// TIA Portal V15.1 export
// export: Created 2024-06-21T08:41:08.5867938Z, ExportSetting WithDefaults, DisplayName Totally Integrated Automation Portal, DisplayVersion V15.1 Update 5, DisplayName TIA Portal Openness, DisplayVersion V15.1 Update 5, DisplayName SINAMICS Startdrive Advanced, DisplayVersion V15.1, DisplayName G130, G150, S120, S150, SINAMICS MV, S210, DisplayVersion V15.1, DisplayName G110M, G120, G120C, G120D, G120P, DisplayVersion V15.1, DisplayName STEP 7 Professional, DisplayVersion V15.1 Update 5, DisplayName STEP 7 Safety, DisplayVersion V15.1, DisplayName WinCC Professional, DisplayVersion V15.1 Update 5, DisplayName SIMATIC Visualization Architect, DisplayVersion V15.1
FUNCTION "LGBJoyStickIAnim" : Void   // FC6612, FBD
TITLE = LIAnimDWord / LGBJoyStickIAnim
{ S7_Optimized_Access := 'TRUE' }
AUTHOR : VCC
FAMILY : Anim
NAME : SIAnim
VERSION : 0.1
// =============================================================================
// Handles the conversion from bits to one Word for simple icon Animation. 
// =============================================================================
// stored: AutoNumber false, IsIECCheckEnabled false, SetENOAutomatically False, UDAEnableTagReadback false
   VAR_INPUT
      I_BtnMiddleAct : Bool;   // Set position / Set Position / Button Middle Active
      I_BtnUpAct : Bool;   // Reset position / Reset Position / Button Up Active
      I_BtnRightAct : Bool;   // Active / Button Right Active
      I_BtnDownAct : Bool;   // ObjectVisible / Button Down Active
      I_BtnLeftAct : Bool;   // Object out of use / Button Left is Active
      I_AnyBtnActive : Bool;   // Any Button Active
      I_OutOfUse : Bool;   // Object out of use
      I_AlarmA : Bool;   // AlarmA
      I_AlarmB : Bool;   // AlarmB
      I_AlarmC : Bool;   // AlarmC
      I_AlarmD : Bool;   // AlarmD
   END_VAR
   VAR_OUTPUT
      H_IAnim : DWord;   // Icon animation Word / Icon Animation
   END_VAR
BEGIN

REGION Network 1: Temporarys output word / **** 1 - Inputs **** Object Out Of Use
   // Object out of use
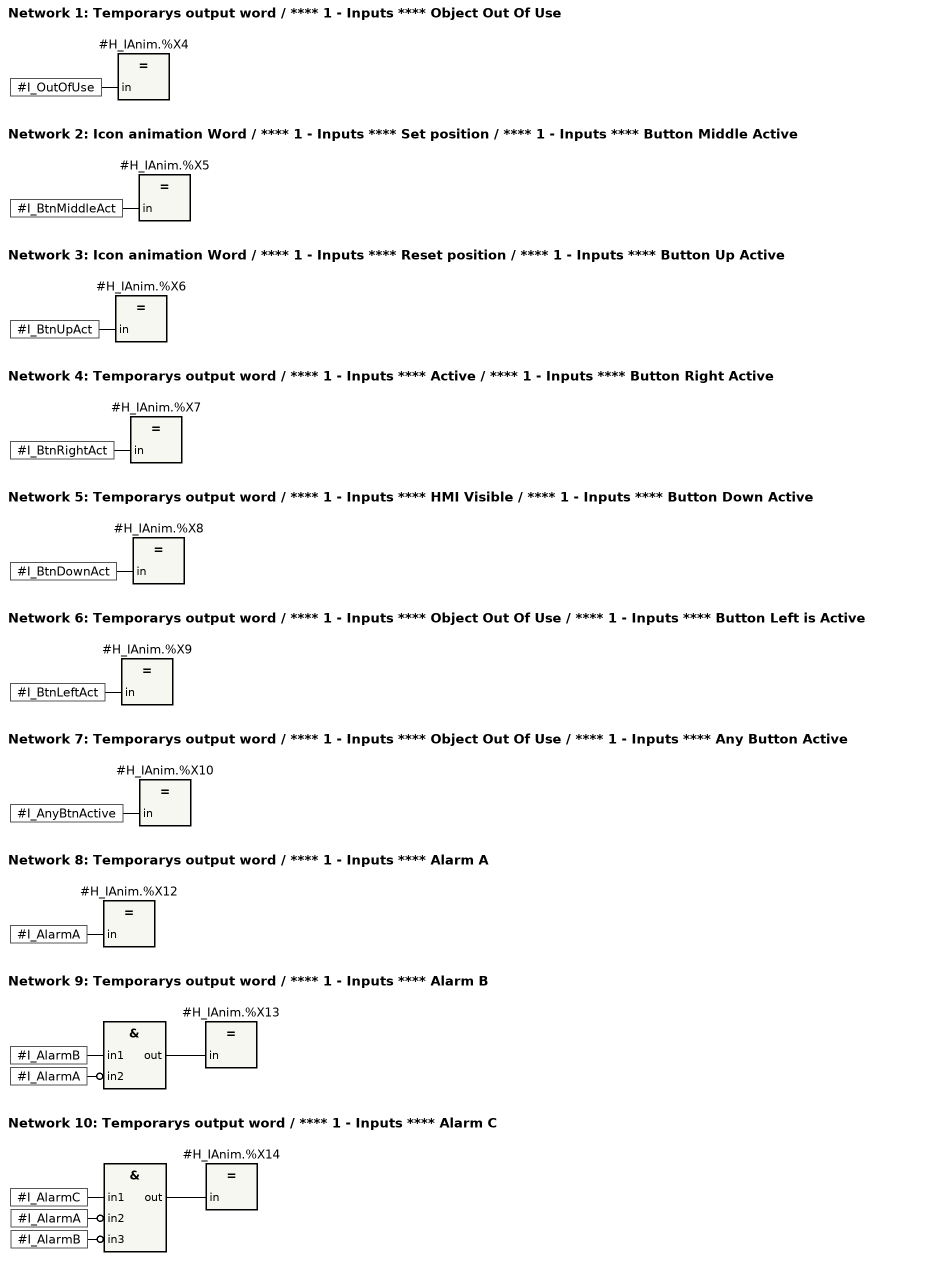
   #H_IAnim.%X4 := #I_OutOfUse;
END_REGION

REGION Network 2: Icon animation Word / **** 1 - Inputs **** Set position / **** 1 - Inputs **** Button Middle Active
   // Set Position
   #H_IAnim.%X5 := #I_BtnMiddleAct;
END_REGION

REGION Network 3: Icon animation Word / **** 1 - Inputs **** Reset position / **** 1 - Inputs **** Button Up Active
   // Reset Position
   #H_IAnim.%X6 := #I_BtnUpAct;
END_REGION

REGION Network 4: Temporarys output word / **** 1 - Inputs **** Active / **** 1 - Inputs **** Button Right Active
   // Active
   #H_IAnim.%X7 := #I_BtnRightAct;
END_REGION

REGION Network 5: Temporarys output word / **** 1 - Inputs **** HMI Visible / **** 1 - Inputs **** Button Down Active
   // HMI Visible
   #H_IAnim.%X8 := #I_BtnDownAct;
END_REGION

REGION Network 6: Temporarys output word / **** 1 - Inputs **** Object Out Of Use / **** 1 - Inputs **** Button Left is Active
   // Object out of use
   #H_IAnim.%X9 := #I_BtnLeftAct;
END_REGION

REGION Network 7: Temporarys output word / **** 1 - Inputs **** Object Out Of Use / **** 1 - Inputs **** Any Button Active
   // Object out of use
   #H_IAnim.%X10 := #I_AnyBtnActive;
END_REGION

REGION Network 8: Temporarys output word / **** 1 - Inputs **** Alarm A
   // Alarm A
   #H_IAnim.%X12 := #I_AlarmA;
END_REGION

REGION Network 9: Temporarys output word / **** 1 - Inputs **** Alarm B
   // Alarm B
   #H_IAnim.%X13 := #I_AlarmB AND NOT #I_AlarmA;
END_REGION

REGION Network 10: Temporarys output word / **** 1 - Inputs **** Alarm C
   // Alarm C
   #H_IAnim.%X14 := #I_AlarmC AND NOT #I_AlarmA AND NOT #I_AlarmB;
END_REGION

REGION Network 11: Temporarys output word / **** 1 - Inputs **** Alarm D
   // Alarm D
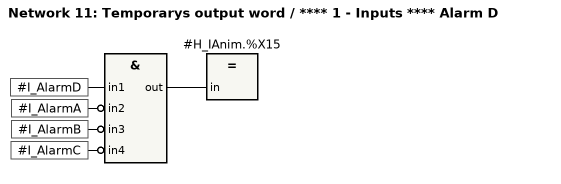
   #H_IAnim.%X15 := #I_AlarmD AND NOT #I_AlarmA AND NOT #I_AlarmB AND NOT #I_AlarmC;
END_REGION
END_FUNCTION
